// TwinCAT 3 PLC project UnitTest
// Title: UnitTest
// Company: Hoox.Software
// Author: Patrick Dressel
// ProjectVersion: 1.0.0
// ProgramVersion: 3.1.4022.6
// libraries:
//   Tc2_Standard, * (Beckhoff Automation GmbH)
//   Tc2_System, * (Beckhoff Automation GmbH)
//   Tc2_Utilities, * (Beckhoff Automation GmbH)
//   Tc3_Module, * (Beckhoff Automation GmbH)
//   Base Interfaces,newest,System
// project tree:
//   Datatypes/Coverage/ ALines_t.TcDUT, EReportType_t.TcDUT (not stored), SCodeCoverage_t.TcDUT (not stored)
//   Datatypes/ EResult_t.TcDUT (not stored), EState_t.TcDUT, IdHandle_t.TcDUT (not stored), ObjectId_t.TcDUT (not stored), SResult_t.TcDUT (not stored), SStatistic_t.TcDUT (not stored), StringHandle_t.TcDUT (not stored), StrMessage_t.TcDUT (not stored), TestCaseHandle_t.TcDUT (not stored), TestSuiteHandle_t.TcDUT
//   Datatypes/Report/ EExportState_t.TcDUT (not stored), ERetCode_t.TcDUT (not stored), NameHandle_t.TcDUT (not stored), PathHandle_t.TcDUT (not stored), StrFileName_t.TcDUT (not stored), StrPathName_t.TcDUT (not stored), TestReportHandle_t.TcDUT, UBaseTypes_t.TcDUT, UTime_t.TcDUT (not stored)
//   / PlcTask.TcTTO (not stored)
//   Source/ FB_Testsuite.TcPOU, FB_UnitTestBase.TcPOU, PRG_UnitTestLib.TcPOU
//   Source/Report/ FB_CoverageFile.TcPOU (not stored), FB_TestReportBase.TcPOU, FB_FileBase.TcPOU, FB_TextReport.TcPOU

// ---- Datatypes/Coverage/ALines_t.TcDUT
TYPE ALines_t : Array[1..1000] of BYTE; END_TYPE

// ---- Datatypes/EState_t.TcDUT
{attribute 'qualified_only'}
{attribute 'strict'}
TYPE EState_t :
(
	eStateInit,
	eStateIdle,
	eStatePrepare,
	eStateExecute,
	eStateCleanUp,
	eStateBuildCoverageFile,
	eStateBuildUnitTestFile,
	eStateReady,
	eStateExport,
	eStateError,
	eStateLicenseError
);
END_TYPE

// ---- Datatypes/Report/TestReportHandle_t.TcDUT
TYPE TestReportHandle_t : Pointer to FB_TestReportBase; END_TYPE

// ---- Datatypes/Report/UBaseTypes_t.TcDUT
TYPE UBaseTypes_t :
UNION
	u8Value 	: USINT;
	s8Value 	: SINT;
	u16Value 	: UINT;
	s16Value 	: INT;
	u32Value 	: UDINT;
	s32Value 	: DINT;
	w16Value    : WORD;
	w32Value    : DWORD;
END_UNION
END_TYPE

// ---- Datatypes/TestSuiteHandle_t.TcDUT
TYPE TestSuiteHandle_t : POINTER TO FB_TestSuite; END_TYPE

// ---- Source/FB_Testsuite.TcPOU
(******************************************************************************
Baustein: FB_Testsuite
Spezifikation: doc/Spezifikation.pdf, Kap. x.y.z
-------------------------------------------------------------------------------
erstellt:
von:
Geändert:
von:
-------------------------------------------------------------------------------
Beschreibung
Dieser Baustein enthält alle zugeordneten Testfälle. Ein Testfall
ist ein abgeleiteter Baustein (FB) von FB_UnitTestBase.

-------------------------------------------------------------------------------
Input
-

Output
-
******************************************************************************)
FUNCTION_BLOCK FB_Testsuite
VAR_INPUT
	i_bStart : BOOL;
END_VAR
VAR_OUTPUT
	o_eState  		: EState_t;
	o_eResult 		: EResult_t;
END_VAR
VAR
	strId			: ObjectId_t;
	strPath			: ObjectId_t;
	bRegistered     : BOOL;
	a_pTest  		: ARRAY [0..255] OF TestCaseHandle_t;
	pTest     		: TestCaseHandle_t;
	u16TestCases  	: UINT;
	u16Index 		: UINT;
	sStatistic 		: SStatistic_t;
END_VAR


	CASE o_eState OF
		
	EState_t.eStateInit:
	
		o_eState 	:= EState_t.eStateError;
		IF bRegistered = TRUE THEN
			o_eState 	:= EState_t.eStateIdle;
		END_IF;
		
	EState_t.eStateIdle:

		u16Index := 0;

		IF i_bStart = TRUE THEN
			logInfo(CONCAT('Run Testsuite ', strId));
			pTest 	 := getFirstTestCase();
			o_eState  := EState_t.eStatePrepare;
			o_eResult := EResult_t.eStatePassed;
		END_IF;

	EState_t.eStatePrepare:
	
		sStatistic.u32Executed  := 0;
		sStatistic.u32Passed 	:= 0;
		sStatistic.u32Failed 	:= 0;
		sStatistic.u32Asserts 	:= 0;

		IF pTest <> 0 THEN
			IF pTest^._prepare() = TRUE THEN
				pTest 	:= getNextTestCase();
			END_IF;
		ELSE
			o_eState := EState_t.eStateExecute;
			pTest 	:= getFirstTestCase();
		END_IF;

	EState_t.eStateExecute:

		IF pTest <> 0 THEN

			IF pTest^.isSkipped() = FALSE THEN

				pTest^.setStartTime();

				IF pTest^._execute() = TRUE THEN
					pTest^.setEndTime();
					sStatistic.u32Executed := sStatistic.u32Executed + 1;	
				
					sStatistic.u32Passed 	:= sStatistic.u32Passed + pTest^.getPassed();
					sStatistic.u32Failed 	:= sStatistic.u32Failed + pTest^.getFailed();
					sStatistic.u32Asserts   := sStatistic.u32Passed + sStatistic.u32Failed;
					
					CASE o_eResult OF 
	
					EResult_t.eStatePassed:
						// Status des letzen Tests übernehmen
						o_eResult := pTest^.o_eResult;
	
					EResult_t.eStateFailed:
						// Status nur übernehmen wenn ein Fatal-Status
						// ermittelt wird und der Test sofort abgebrochen
						// werden soll.
						IF pTest^.o_eResult = EResult_t.eStateFailedFatal THEN
							o_eResult := pTest^.o_eResult;
							o_eState  := EState_t.eStateCleanUp;
							pTest 	  := getFirstTestCase();	
						END_IF;
	
					EResult_t.eStateFailedFatal:
	
						o_eState := EState_t.eStateCleanUp;
						pTest 	:= getFirstTestCase();					
	
					END_CASE;
	
					IF o_eResult <> EResult_t.eStateFailedFatal THEN
						pTest 	 := getNextTestCase();
					END_IF;
	
				END_IF;
			ELSE
				pTest 	 := getNextTestCase();
			END_IF;
		ELSE
			o_eState := EState_t.eStateCleanUp;
			pTest 	:= getFirstTestCase();
		END_IF;

	ESTate_t.eStateCleanUp:

		IF pTest <> 0 THEN
			IF pTest^._cleanup() = TRUE THEN
				pTest 	:= getNextTestCase();
			END_IF;
		ELSE
			o_eState := EState_t.eStateReady;
		END_IF;
		
	ESTate_t.eStateReady:
	
		IF i_bStart = FALSE THEN
			o_eState := EState_t.eStateIdle;
		END_IF
		
	ESTate_t.eStateError:	
		
		// wenn wir hier rauskommen ist was dummes passiert
		
	ELSE
		
		o_eState := EState_t.eStateError;
		
	END_CASE;
	
	
	
	
	
	
//

(******************************************************************************
Baustein: FB_Testsuite.addTestcase
Spezifikation: doc/Spezifikation.pdf, Kap. x.y.z
-------------------------------------------------------------------------------
erstellt:
von:
Geändert:
von:
-------------------------------------------------------------------------------
Beschreibung
Diese Methode

-------------------------------------------------------------------------------
Input
i_pTestCase

Output
-
******************************************************************************)
{attribute 'hide'} 
METHOD PUBLIC addTestcase : BOOL
VAR_INPUT
	i_pTestCase : TestCaseHandle_t;
END_VAR

	addTestcase := FALSE;

	IF 	i_pTestCase  <> 0   AND 
		u16TestCases <  255 THEN
		
		a_pTest[u16TestCases] := i_pTestCase;
		
		u16TestCases := u16TestCases +1;
		
		sStatistic.u32TestCases := sStatistic.u32TestCases + 1;
		
		addTestcase := true;
	END_IF
END_METHOD

(******************************************************************************
Baustein: FB_Testsuite.FB_init
Spezifikation: doc/Spezifikation.pdf, Kap. x.y.z
-------------------------------------------------------------------------------
erstellt:
von:
Geändert:
von:
-------------------------------------------------------------------------------
Beschreibung
Diese Methode

-------------------------------------------------------------------------------
Input
i_pTestCase

Output
-
******************************************************************************)
{attribute 'hide'} 
METHOD FB_init : BOOL
VAR_INPUT
	bInitRetains 	: BOOL; // if TRUE, the retain variables are initialized (warm start / cold start)
	bInCopyCode 	: BOOL;  // if TRUE, the instance afterwards gets moved into the copy code (online change)
	i_strId	  		: ObjectId_t;
	i_strPath		: ObjectId_t;
END_VAR

	strId 	:= i_StrId;
	strPath := i_strPath;
	register();
END_METHOD

(******************************************************************************
Baustein: FB_Testsuite.getExecuted
Spezifikation: doc/Spezifikation.pdf, Kap. x.y.z
-------------------------------------------------------------------------------
erstellt:
von:
Geändert:
von:
-------------------------------------------------------------------------------
Beschreibung
Diese Methode

-------------------------------------------------------------------------------
Input
-

Output
-
******************************************************************************)
{attribute 'hide'} 
METHOD PUBLIC getExecuted : UDINT
VAR_INPUT
END_VAR

	getExecuted := sStatistic.u32Executed;
END_METHOD

(******************************************************************************
Baustein: FB_Testsuite.getFailed
Spezifikation: doc/Spezifikation.pdf, Kap. x.y.z
-------------------------------------------------------------------------------
erstellt:
von:
Geändert:
von:
-------------------------------------------------------------------------------
Beschreibung
Diese Methode

-------------------------------------------------------------------------------
Input
-

Output
-
******************************************************************************)
{attribute 'hide'} 
METHOD PUBLIC getFailed : UDINT
VAR_INPUT
END_VAR

	getFailed := sStatistic.u32Failed;
END_METHOD

(******************************************************************************
Baustein: FB_Testsuite.getFirstTestCase
Spezifikation: doc/Spezifikation.pdf, Kap. x.y.z
-------------------------------------------------------------------------------
erstellt:
von:
Geändert:
von:
-------------------------------------------------------------------------------
Beschreibung
Diese Methode

-------------------------------------------------------------------------------
Input
-

Output
-
******************************************************************************)
{attribute 'hide'} 
METHOD PUBLIC getFirstTestCase : TestCaseHandle_t
VAR_INPUT
END_VAR

	u16Index := 0;
	getFirstTestCase := a_pTest[0];
END_METHOD

(******************************************************************************
Baustein: FB_Testsuite.getId
Spezifikation: doc/Spezifikation.pdf, Kap. x.y.z
-------------------------------------------------------------------------------
erstellt:
von:
Geändert:
von:
-------------------------------------------------------------------------------
Beschreibung
Diese Methode

-------------------------------------------------------------------------------
Input
-

Output
-
******************************************************************************)
{attribute 'hide'} 
METHOD PUBLIC getId : STRING
VAR_INPUT
END_VAR

	getId := strId;
END_METHOD

(******************************************************************************
Baustein: FB_Testsuite.getNextTestCase
Spezifikation: doc/Spezifikation.pdf, Kap. x.y.z
-------------------------------------------------------------------------------
erstellt:
von:
Geändert:
von:
-------------------------------------------------------------------------------
Beschreibung
Diese Methode

-------------------------------------------------------------------------------
Input
-

Output
-
******************************************************************************)
{attribute 'hide'} 
METHOD PUBLIC getNextTestCase : TestCaseHandle_t
VAR_INPUT
END_VAR

	getNextTestCase := 0;
	u16Index 		 := u16Index + 1;

	IF u16Index < u16TestCases THEN
		getNextTestCase := a_pTest[u16Index];
	END_IF;
END_METHOD

(******************************************************************************
Baustein: FB_Testsuite.getNoOfAsserts
Spezifikation: doc/Spezifikation.pdf, Kap. x.y.z
-------------------------------------------------------------------------------
erstellt:
von:
Geändert:
von:
-------------------------------------------------------------------------------
Beschreibung
Diese Methode

-------------------------------------------------------------------------------
Input
-

Output
-
******************************************************************************)
{attribute 'hide'} 
METHOD PUBLIC getNoOfAsserts : UDINT
VAR_INPUT
END_VAR

	getNoOfAsserts := sStatistic.u32Asserts;
END_METHOD

(******************************************************************************
Baustein: FB_Testsuite.getNoOfTests
Spezifikation: doc/Spezifikation.pdf, Kap. x.y.z
-------------------------------------------------------------------------------
erstellt:
von:
Geändert:
von:
-------------------------------------------------------------------------------
Beschreibung
Diese Methode

-------------------------------------------------------------------------------
Input
-

Output
-
******************************************************************************)
{attribute 'hide'} 
METHOD PUBLIC getNoOfTests : UDINT
VAR_INPUT
END_VAR

	getNoOfTests := sStatistic.u32TestCases;
END_METHOD

(******************************************************************************
Baustein: FB_Testsuite.getPassed
Spezifikation: doc/Spezifikation.pdf, Kap. x.y.z
-------------------------------------------------------------------------------
erstellt:
von:
Geändert:
von:
-------------------------------------------------------------------------------
Beschreibung
Diese Methode

-------------------------------------------------------------------------------
Input
-

Output
-
******************************************************************************)
{attribute 'hide'} 
METHOD PUBLIC getPassed : UDINT
VAR_INPUT
END_VAR

	getPassed := sStatistic.u32Passed;
END_METHOD

{attribute 'hide'} 
METHOD PUBLIC getPath : ObjectId_t
VAR_INPUT
END_VAR

	getPath := strPath;
END_METHOD

(******************************************************************************
Baustein: FB_Testsuite.logInfo
Spezifikation: doc/Spezifikation.pdf, Kap. x.y.z
-------------------------------------------------------------------------------
erstellt:
von:
Geändert:
von:
-------------------------------------------------------------------------------
Beschreibung
Diese Methode

-------------------------------------------------------------------------------
Input
i_strMessage

Output
-
******************************************************************************)
{attribute 'hide'} 
METHOD PROTECTED logInfo : BOOL
VAR_INPUT
	i_strMessage : StrMessage_t;
END_VAR

	ADSLOGSTR(msgCtrlMask 	:= ADSLOG_MSGTYPE_HINT , 
			  msgFmtStr 	:= i_strMessage, 
			  strArg 		:= '');
END_METHOD

(******************************************************************************
Baustein: FB_Testsuite.register
Spezifikation: doc/Spezifikation.pdf, Kap. x.y.z
-------------------------------------------------------------------------------
erstellt:
von:
Geändert:
von:
-------------------------------------------------------------------------------
Beschreibung
Diese Methode

-------------------------------------------------------------------------------
Input
-

Output
-
******************************************************************************)
{attribute 'hide'} 
METHOD PROTECTED register : BOOL
VAR_INPUT
END_VAR

	bRegistered := PRG_UnitTestLib.addTestSuite(this);
END_METHOD

END_FUNCTION_BLOCK

// ---- Source/PRG_UnitTestLib.TcPOU
(******************************************************************************
Baustein: PRG_TestLibrary
Spezifikation: doc/Spezifikation.pdf, Kap. x.y.z
-------------------------------------------------------------------------------
erstellt:
von:
Geändert:
von:
-------------------------------------------------------------------------------
Beschreibung
Dieser Baustein etnhält alle Testsuites und führt diese aus.

-------------------------------------------------------------------------------
Input
	i_bStart : mit positiver Flanke werden die registrierten Testsuites ausgeführt

Output
	o_eState  		: EState_t;
	o_eResult 		: EResult_t;
	o_sStatistic	: SStatistic_t;
******************************************************************************)
{attribute 'global_init_slot' := '41000'}
PROGRAM PRG_UnitTestLib
VAR_INPUT
	i_bStart : BOOL;
END_VAR
VAR_OUTPUT
	o_eState  		: EState_t;
	o_eResult 		: EResult_t;
	o_sStatistic	: SStatistic_t;
END_VAR
VAR
	a_pTestSuite 	: ARRAY [0..255] OF TestSuiteHandle_t;
	u16TestSuites 	: UINT;
	u16Index	  	: UINT;
	pActTestSuite 	: TestSuiteHandle_t;
	pTestReport		: POINTER TO FB_TestReportBase;
	eRetCode 		: ERetCode_t;

	fbSystemTime 	: FB_LocalSystemTime;
	
	fbLicense 		: FB_CheckLicense;
	
	
	fbCoverage 		: FB_CoverageFile;
	fbUnittest 		: FB_CoverageFile;
	u16PouIdx  		: UINT;
	u16LineIdx 		: UINT;
	u16ReportState  : UINT;
	u16TestSuitIdx	: UINT;
	sCodeCoverage	: SCodeCoverage_t;
	pTestCase  		: TestCaseHandle_t;
END_VAR


	fbSystemTime(bEnable := TRUE, dwCycle := 5);

	fbCoverage();

	fbUnittest();

	CASE o_eState OF 
	
	EState_t.eStateInit:	

		//IF checkLicense() = ERetCode_t.eRetDone THEN
			
			IF i_bStart = FALSE THEN 
				o_eState := EState_t.eStateIdle; 
			END_IF
			
		//END_IF;
	
	EState_t.eStateIdle:
	
		IF i_bStart = TRUE THEN
			logInfo('+++++++++++++ Testbeginn ++++++++++++++');
			o_eState := EState_t.eStatePrepare;
		END_IF
	
	EState_t.eStatePrepare:
		
		o_eResult 	  				:= EResult_t.eStatePassed;
		o_sStatistic.u32Executed 	:= 0;
		o_sStatistic.u32TestCases	:= 0;
		o_sStatistic.u32Asserts  	:= 0;
		o_sStatistic.u32Passed   	:= 0;
		o_sStatistic.u32Failed	 	:= 0;	

		pActTestSuite := getFirstTestSuite();
		
		IF pActTestSuite      <> 0   THEN
			o_eState := EState_t.eStateExecute;
		ELSE
			o_eState := EState_t.eStateError;	
		END_IF
	
	EState_t.eStateExecute:
	
		pActTestSuite^(i_bStart := TRUE);
	
		IF pActTestSuite^.o_eState = EState_t.eStateReady THEN
			
			IF pActTestSuite^.o_eResult = EResult_t.eStateFailed THEN
				o_eResult := EResult_t.eStateFailed;
			END_IF
			
			pActTestSuite^(i_bStart := FALSE);
			
			o_eState := EState_t.eStateCleanUp;
			
			o_sStatistic.u32Executed 	:= o_sStatistic.u32Executed  + pActTestSuite^.getExecuted();
			o_sStatistic.u32TestCases	:= o_sStatistic.u32TestCases + pActTestSuite^.getNoOfTests(); 
			o_sStatistic.u32Asserts  	:= o_sStatistic.u32Asserts   + pActTestSuite^.getNoOfAsserts();
			o_sStatistic.u32Passed   	:= o_sStatistic.u32Passed    + pActTestSuite^.getPassed();
			o_sStatistic.u32Failed	 	:= o_sStatistic.u32Failed    + pActTestSuite^.getFailed();
		END_IF
	
	EState_t.eStateCleanUp:
	
		IF pActTestSuite^.o_eResult = EResult_t.eStateFailedFatal THEN
			o_eResult := EResult_t.eStateFailedFatal;
			o_eState  := EState_t.eStateBuildCoverageFile;
		ELSE
			
			pActTestSuite := getNextTestSuite();
						
			IF pActTestSuite <> 0 THEN
				o_eState := EState_t.eStateExecute;
			ELSE
				o_eState := EState_t.eStateBuildCoverageFile;
				logInfo('+++++++++++++ Test Ende ++++++++++++++');
			END_IF		
			
		END_IF

	EState_t.eStateBuildCoverageFile:

		IF createReport(EReporttype_t.eCoverageReport) = ERetCode_t.eRetDone THEN
			o_eState := EState_t.eStateBuildUnitTestFile;
		END_IF;

	EState_t.eStateBuildUnitTestFile:

		IF createReport(EReporttype_t.eUnitTestReport) = ERetCode_t.eRetDone THEN
			o_eState := EState_t.eStateReady;
		END_IF;

	EState_t.eStateReady:

		IF i_bStart = FALSE THEN
			o_eState := EState_t.eStateExport;
		END_IF

	EState_t.eStateExport:

		IF createReport(EReporttype_t.eExternalReport) = ERetCode_t.eRetDone THEN
			o_eState := EState_t.eStateIdle;
		END_IF;

	EState_t.eStateError,
	EState_t.eStateLicenseError:
	
		o_eState := EState_t.eStateError;

	END_CASE

(******************************************************************************
Baustein: PRG_UnitTestLib.addTestReport
Spezifikation: doc/Spezifikation.pdf, Kap. x.y.z
-------------------------------------------------------------------------------
erstellt:
von:
Geändert:
von:
-------------------------------------------------------------------------------
Beschreibung
Diese Methode

-------------------------------------------------------------------------------
Input
i_pTestReport

Output
-
******************************************************************************)
{attribute 'hide'} 
METHOD PUBLIC addTestReport : BOOL
VAR_INPUT
	i_pTestReport : TestReportHandle_t;
END_VAR

	pTestReport := i_pTestReport;
END_METHOD

(******************************************************************************
Baustein: PRG_UnitTestLib.addTestSuite
Spezifikation: doc/Spezifikation.pdf, Kap. x.y.z
-------------------------------------------------------------------------------
erstellt:
von:
Geändert:
von:
-------------------------------------------------------------------------------
Beschreibung
Diese Methode

-------------------------------------------------------------------------------
Input
i_pTestSuite

Output
-
******************************************************************************)
{attribute 'hide'} 
METHOD PUBLIC addTestSuite : BOOL
VAR_INPUT
	i_pTestSuite : TestSuiteHandle_t;
END_VAR

	addTestSuite := FALSE;

	IF 	i_pTestSuite  <> 0   AND 
		u16TestSuites <  255 THEN
		
		a_pTestSuite[u16TestSuites] := i_pTestSuite;
		
		u16TestSuites := u16TestSuites +1;
	
		o_sStatistic.u32TestSuites := o_sStatistic.u32TestSuites + 1;
		o_sStatistic.u32TestCases  := o_sStatistic.u32TestCases + i_pTestSuite^.sStatistic.u32TestCases;
		
		addTestSuite := TRUE;
	END_IF
END_METHOD

(******************************************************************************
Baustein: PRG_UnitTestLib.checkLicense
Spezifikation: doc/Spezifikation.pdf, Kap. x.y.z
-------------------------------------------------------------------------------
erstellt:
von:
Geändert:
von:
-------------------------------------------------------------------------------
Beschreibung
Diese Methode

-------------------------------------------------------------------------------
Input
-

Output
-
******************************************************************************)
{attribute 'hide'} 
METHOD checkLicense : ERetCode_t
VAR_INPUT
END_VAR

	checkLicense := ERetCode_t.eRetBusy;
	
	fbLicense(bExecute    := TRUE, 
		  stLicenseId := STRING_TO_GUID('994D9F0C-F802-4000-8582-229354A3CA39'));
			  
	IF fbLicense.bBusy =  FALSE THEN
		IF fbLicense.stCheckLicense.eResult = E_LHR_LicenseOK THEN
			checkLicense := ERetCode_t.eRetDone;
		ELSE
			checkLicense := ERetCode_t.eRetFailed;	
		END_IF
	END_IF;
END_METHOD

{attribute 'hide'} 
METHOD PRIVATE createReport : ERetCode_t
VAR_INPUT
	i_eReporttype : EReportType_t;
END_VAR
VAR
	eRetcode : ERetCode_t;
	u32Temp : UDINT;
END_VAR

	createReport := ERetCode_t.eRetBusy;

	CASE u16ReportState OF

	0: 
		IF i_eReporttype = EReportType_t.eCoverageReport THEN
			u16ReportState := 10;
		END_IF;

		IF i_eReporttype = EReportType_t.eUnitTestReport THEN
			u16ReportState := 20;
		END_IF;

		IF i_eReporttype = EReportType_t.eExternalReport THEN
			u16ReportState := 100;
		END_IF;

// +++++++++++++++++++++++++++++++++++++++++++++++++++++++++++
//
// Export Codeabdeckung
// 
// +++++++++++++++++++++++++++++++++++++++++++++++++++++++++++
	10:
		eRetcode := fbCoverage.open('C:\Users\Administrator\Desktop\TestResult\', 'Coverage.xml');

		IF eRetcode = ERetCode_t.eRetDone THEN

			u16ReportState := 11;

		ELSIF eRetcode = ERetCode_t.eRetFailed THEN

			logError('createReport Coverage.xml : Datei nicht geöffnet');
			u16ReportState := 12;

		END_IF;		

	11:

		fbCoverage.addString('<?xml version="1.0" ?>');
		fbCoverage.addCrlf();

		fbCoverage.addString('<Result>');
		fbCoverage.addCrlf();

		FOR u16PouIdx := 1 TO sCodeCoverage.u16MaxIndex DO

			fbCoverage.addString('<POU Id="');
			fbCoverage.addValue(u16PouIdx);
			fbCoverage.addString('">');
			fbCoverage.addCrlf();

			FOR u16LineIdx := 1 TO 1000 DO

				IF sCodeCoverage.aPou[u16PouIdx][u16LineIdx] > 0 THEN

					fbCoverage.addString('<Line Nb="');
					fbCoverage.addValue(u16LineIdx);

					fbCoverage.addString('" Count="');
					fbCoverage.addValue(sCodeCoverage.aPou[u16PouIdx][u16LineIdx]);
					
					fbCoverage.addString('"/>');
					fbCoverage.addCrlf();

				END_IF;

			END_FOR;

			fbCoverage.addString('</POU>');
			fbCoverage.addCrlf();

		END_FOR;

		fbCoverage.addString('</Result>');
		fbCoverage.addCrlf();
		u16ReportState := 12;


	12:

		IF fbCoverage.o_bOpen  = TRUE AND 
		   fbCoverage.o_bEmpty = TRUE THEN
			fbCoverage.close();
		END_IF;

		IF fbCoverage.o_bOpen  = FALSE THEN
			createReport 	:= ERetCode_t.eRetDone;
		END_IF;

// +++++++++++++++++++++++++++++++++++++++++++++++++++++++++++
//
// Export Unittest Ergebnisse
// 
// +++++++++++++++++++++++++++++++++++++++++++++++++++++++++++
	20:		

		eRetcode := fbUnitTest.open('C:\Users\Administrator\Desktop\TestResult\', 'Unittest.xml');

		IF eRetcode = ERetCode_t.eRetDone THEN

			u16ReportState := 21;

		ELSIF eRetcode = ERetCode_t.eRetFailed THEN

			logError('createReport Unittest.xml : Datei nicht geöffnet');
			u16ReportState := 22;

		END_IF;	

	21:

		u16TestSuitIdx := 0;

		fbUnitTest.addString('<?xml version="1.0" ?>');
		fbUnitTest.addCrlf();

		fbUnitTest.addString('<testsuites>');
		fbUnitTest.addCrlf();

		pActTestSuite := getFirstTestSuite();

		WHILE (pActTestSuite <> 0) DO

			u16TestSuitIdx := u16TestSuitIdx+1;

			fbUnitTest.addString('<testsuite');
			fbUnitTest.addString(' name="');
			fbUnitTest.addString(pActTestSuite^.getId());
			fbUnitTest.addString('" tests="');
			u32Temp := pActTestSuite^.getNoOfTests();
			fbUnitTest.addValue(u32Temp);
			fbUnitTest.addString('" disabled="');
			u32Temp := 0;
			fbUnitTest.addValue(u32Temp);
			fbUnitTest.addString('" errors="');
			fbUnitTest.addValue(u32Temp);
			fbUnitTest.addString('" failures="');
			u32Temp := pActTestSuite^.getFailed();
			fbUnitTest.addValue(u32Temp);
			fbUnitTest.addString('" hostname="');
			fbUnitTest.addString('" id="');
			fbUnitTest.addvalue(u16TestSuitIdx);
			fbUnitTest.addString('" package="');
			fbUnitTest.addString(pActTestSuite^.getPath());
			fbUnitTest.addString('">');
			fbUnitTest.addCrlf();

			pTestCase := pActTestSuite^.getFirstTestCase();

			WHILE (pTestCase <> 0) DO

				fbUnitTest.addString('<testcase');
				fbUnitTest.addString(' name="');
				fbUnitTest.addString(pTestCase^.getId());
				fbUnitTest.addString('" assertions="');
				u32Temp := pTestCase^.getFailed() + pTestCase^.getPassed();
				fbUnitTest.addValue(u32Temp);
				fbUnitTest.addString('" classname="');
				fbUnitTest.addString(pTestCase^.getPath());
				fbUnitTest.addString(pTestCase^.getClassName());
				fbUnitTest.addString('" time="');
				u32Temp := pTestCase^.getTime();
				fbUnitTest.addTimeMs(u32Temp);
				fbUnitTest.addString('">');
				fbUnitTest.addCrlf();

				CASE pTestCase^.o_eResult OF

				EResult_t.eStatePassed :

					fbUnitTest.addString('<passed/>');

				EResult_t.eStateFailed, 
				EResult_t.eStateFailedFatal :
			
					fbUnitTest.addString('<failure/>');

				EResult_t.eStateSkipped:

					fbUnitTest.addString('<skipped/>');

				END_CASE;
				
				fbUnitTest.addCrlf();	

				fbUnitTest.addString('</testcase>');
				fbUnitTest.addCrlf();		

				pTestCase := pActTestSuite^.getNextTestCase();
		
			END_WHILE

			fbUnitTest.addString('</testsuite>');
			fbUnitTest.addCrlf();	

			pActTestSuite := getNextTestSuite();

		END_WHILE

		fbUnitTest.addString('</testsuites>');
		fbUnitTest.addCrlf();

		u16ReportState := 22;

	22:
		IF fbUnitTest.o_bOpen  = TRUE AND 
		   fbUnitTest.o_bEmpty = TRUE THEN
			fbUnitTest.close();
		END_IF;

		IF fbUnitTest.o_bOpen  = FALSE THEN
			createReport 	:= ERetCode_t.eRetDone;
		END_IF;

// +++++++++++++++++++++++++++++++++++++++++++++++++++++++++++
//
//
// 
// +++++++++++++++++++++++++++++++++++++++++++++++++++++++++++
	100:

		IF pTestReport <> 0 THEN
			
			createReport := pTestReport^.create();		
			
		ELSE

			createReport := ERetCode_t.eRetDone;

		END_IF;

	ELSE
		createReport := ERetCode_t.eRetFailed;
	END_CASE;

	IF createReport = ERetCode_t.eRetDone THEN
		u16ReportState := 0;
	END_IF;
















(**)
END_METHOD

(******************************************************************************
Baustein: PRG_UnitTestLib.getFirstTestSuite
Spezifikation: doc/Spezifikation.pdf, Kap. x.y.z
-------------------------------------------------------------------------------
erstellt:
von:
Geändert:
von:
-------------------------------------------------------------------------------
Beschreibung
Diese Methode

-------------------------------------------------------------------------------
Input
-

Output
-
******************************************************************************)
{attribute 'hide'} 
METHOD PRIVATE getFirstTestSuite : TestSuiteHandle_t
VAR_INPUT
END_VAR

	u16Index := 0;
	getFirstTestSuite := a_pTestSuite[0];
END_METHOD

(******************************************************************************
Baustein: PRG_UnitTestLib.getNextTestSuite
Spezifikation: doc/Spezifikation.pdf, Kap. x.y.z
-------------------------------------------------------------------------------
erstellt:
von:
Geändert:
von:
-------------------------------------------------------------------------------
Beschreibung
Diese Methode

-------------------------------------------------------------------------------
Input
-

Output
-
******************************************************************************)
{attribute 'hide'} 
METHOD PRIVATE getNextTestSuite : TestSuiteHandle_t
VAR_INPUT
END_VAR

	getNextTestSuite := 0;
	u16Index 		 := u16Index + 1;

	IF u16Index < u16TestSuites THEN
		getNextTestSuite := a_pTestSuite[u16Index];
	END_IF;
END_METHOD

(******************************************************************************
Baustein: PRG_UnitTestLib.getTime
Spezifikation: doc/Spezifikation.pdf, Kap. x.y.z
-------------------------------------------------------------------------------
erstellt:
von:
Geändert:
von:
-------------------------------------------------------------------------------
Beschreibung
Diese Methode

-------------------------------------------------------------------------------
Input
-

Output
-
******************************************************************************)
{attribute 'hide'} 
METHOD getTime : TimeStruct
VAR_INPUT
END_VAR
VAR
END_VAR

	getTime := fbSystemTime.systemTime;
END_METHOD

{attribute 'hide'} 
METHOD PUBLIC LineCovered : BOOL
VAR_INPUT
	u16Pou  : UINT;
	u16Line : UINT;
END_VAR

	LineCovered := TRUE;
	
	IF o_eState = EState_t.eStateExecute THEN

		IF (u16Pou  > 0 AND u16Pou  <= 2000) AND
           (u16Line > 0 AND u16Line <= 1000) THEN

			IF u16Pou > sCodeCoverage.u16MaxIndex THEN
				sCodeCoverage.u16MaxIndex := u16Pou;
			END_IF;

			IF sCodeCoverage.aPou[u16Pou][u16Line] < 255 THEN
				sCodeCoverage.aPou[u16Pou][u16Line] := sCodeCoverage.aPou[u16Pou][u16Line]+1;
			END_IF;
		END_IF;

	END_IF;
END_METHOD

(******************************************************************************
Baustein: PRG_UnitTestLib.logError
Spezifikation: doc/Spezifikation.pdf, Kap. x.y.z
-------------------------------------------------------------------------------
erstellt:
von:
Geändert:
von:
-------------------------------------------------------------------------------
Beschreibung
Diese Methode

-------------------------------------------------------------------------------
Input
i_strMessage

Output
-
******************************************************************************)
{attribute 'hide'} 
METHOD PROTECTED logError : BOOL
VAR_INPUT
	i_strMessage : StrMessage_t;
END_VAR

	ADSLOGSTR(msgCtrlMask 	:= ADSLOG_MSGTYPE_ERROR , 
			  msgFmtStr 	:= i_strMessage, 
			  strArg 		:= '');
END_METHOD

(******************************************************************************
Baustein: PRG_UnitTestLib.logInfo
Spezifikation: doc/Spezifikation.pdf, Kap. x.y.z
-------------------------------------------------------------------------------
erstellt:
von:
Geändert:
von:
-------------------------------------------------------------------------------
Beschreibung
Diese Methode

-------------------------------------------------------------------------------
Input
i_strMessage

Output
-
******************************************************************************)
{attribute 'hide'} 
METHOD PUBLIC logInfo : BOOL
VAR_INPUT
	i_strMessage : StrMessage_t;
END_VAR

	ADSLOGSTR(msgCtrlMask 	:= ADSLOG_MSGTYPE_HINT , 
			  msgFmtStr 	:= i_strMessage, 
			  strArg 		:= '');
END_METHOD

END_PROGRAM

// ---- Source/Report/FB_TestReportBase.TcPOU
(******************************************************************************
Baustein: FB_TestReportBase
Spezifikation: doc/Spezifikation.pdf, Kap. x.y.z
-------------------------------------------------------------------------------
erstellt:
von:
Geändert:
von:
-------------------------------------------------------------------------------
Beschreibung
Dieser Baustein enthält alle zugeordneten Testfälle. Ein Testfall
ist ein abgeleiteter Baustein (FB) von FB_UnitTestBase.

-------------------------------------------------------------------------------
Input
-

Output
-
******************************************************************************)
FUNCTION_BLOCK FB_TestReportBase
VAR_INPUT
END_VAR
VAR_OUTPUT
END_VAR
VAR
	strBuffer   : STRING(255);
	fbOpen      : FB_FileOpen;
	fbClose     : FB_FileClose;
	fbWrite	    : FB_FileWrite;
	strFileName : StrFileName_t;
	strFilePath : StrPathName_t;
	
	eState 		: EExportState_t;
	u32Line     : UDINT;
	
	sStatistic  : SStatistic_t;

	trgOpen 	: F_TRIG;
	trgWrite 	: F_TRIG;
	trgClose 	: F_TRIG;
END_VAR

METHOD PROTECTED addCrlf : BOOL
VAR_INPUT
END_VAR
VAR
END_VAR
   
	strBuffer := CONCAT(strBuffer, '$R$N');
END_METHOD

METHOD PROTECTED addDate : ERetCode_t
VAR_INPUT
	i_sDate : TIMESTRUCT;
END_VAR

   	addDate := ERetcode_t.eRetDone;

   	addValue(i_sDate.wDay);
   	addString('.');
   	addValue(i_sDate.wMonth);
   	addString('.');
    addValue(i_sDate.wYear);
    addString(' ');
END_METHOD

METHOD PROTECTED addString : ERetCode_t
VAR_INPUT
	i_strData : STRING(255);
END_VAR

	strBuffer :=  concat(strBuffer, i_strData);

	addString := ERetcode_t.eRetDone;
END_METHOD

METHOD PROTECTED addTime : ERetCode_t
VAR_INPUT
	i_sTime : TIMESTRUCT;
END_VAR

	addTime := ERetcode_t.eRetDone;
	
   	addValue(i_sTime.wHour);
   	addString('.');
   	addValue(i_sTime.wMinute);
  	addString('.');
   	addValue(i_sTime.wSecond);
   	addString(' ');
END_METHOD

METHOD PROTECTED addValue : ERetCode_t
VAR_INPUT
	i_anyValue : ANY;
END_VAR
VAR
	uValue : UBaseTypes_t;
END_VAR

	addValue  := ERetcode_t.eRetDone;
	
	IF i_anyValue.pValue = 0 THEN
		addValue  := ERetcode_t.eRetFailed;
		RETURN;
	END_IF

	MEMCPY(ADR(uValue),i_anyValue.pValue, TO_UDINT(i_anyValue.diSize)); 

	CASE i_anyValue.TypeClass OF

	IBaseLibrary.TYPE_SINT:

		addString(SINT_TO_STRING(uValue.s8Value));

	//IBaseLibrary.TYPE_BYTE:
	IBaseLibrary.TYPE_USINT:

		addString(USINT_TO_STRING(uValue.u8Value));

	IBaseLibrary.TYPE_INT:

		addString(INT_TO_STRING(uValue.s16Value));

	IBaseLibrary.TYPE_DINT:

		addString(DINT_TO_STRING(uValue.s32Value));

	IBaseLibrary.TYPE_UINT:

		addString(UINT_TO_STRING(uValue.u16Value));

	IBaseLibrary.TYPE_UDINT:

		addString(UDINT_TO_STRING(uValue.u32Value));

	IBaseLibrary.TYPE_WORD:

		addString(WORD_TO_STRING(uValue.w16Value));

	IBaseLibrary.TYPE_DWORD:

		addString(DWORD_TO_STRING(uValue.w32Value));

	ELSE
		ADSLOGSTR(msgCtrlMask 	:= ADSLOG_MSGTYPE_ERROR , 
				  msgFmtStr 	:= 'TestReportBase.AddValue: Unbekannter Datentyp!', 
				  strArg 		:= '');
	END_CASE;
END_METHOD

(******************************************************************************
Baustein: FB_TestReportBase.BuildFile
Spezifikation: doc/Spezifikation.pdf, Kap. x.y.z
-------------------------------------------------------------------------------
erstellt:
von:
Geändert:
von:
-------------------------------------------------------------------------------
Beschreibung
Diese Methode muss vom ableitenden Baustein überschrieben werden und
wird von der Basisklasse aus aufgerufen wenn der Report erstellt werden
soll.

-------------------------------------------------------------------------------
Input
-

Output
-
******************************************************************************)
METHOD PROTECTED BuildFile : ERetCode_t
VAR_INPUT
	i_u32Line : UDINT;
END_VAR
END_METHOD

METHOD PROTECTED clearBuffer : ERetCode_t
VAR_INPUT
END_VAR

	clearBuffer := ERetCode_t.eRetDone;
	
	strBuffer := '';
END_METHOD

METHOD PROTECTED Close : ERetCode_t
VAR_INPUT
END_VAR

	Close := ERetCode_t.eRetFailed;
	
	fbClose.hFile 		:= fbOpen.hFile;
	fbClose.bExecute 	:= TRUE; 

	IF trgClose.Q = TRUE THEN
		Close := ERetCode_t.eRetDone;
		fbClose.bExecute  := FALSE;		
	ELSE	
		Close := ERetCode_t.eRetBusy;
	END_IF;	
	
	IF fbClose.bError = TRUE THEN
		Close := eRetCode_t.eRetFailed;
	END_IF;
END_METHOD

METHOD PUBLIC create : ERetCode_t;
VAR_INPUT
END_VAR
VAR
	eRetCode : ERetCode_t;
END_VAR

	create := ERetCode_t.eRetBusy;

	fbOpen();
	fbWrite();
	fbClose();

	trgOpen(CLK := fbOpen.bBusy);
	trgWrite(CLK := fbWrite.bBusy);
	trgClose(CLK := fbClose.bBusy);
	
	CASE eState OF
	
	EExportState_t.eExportIdle:
	
		eState := EExportState_t.eExportOpen;
	
	EExportState_t.eExportOpen:
	
		eRetCode 	:= Open();
		u32Line  	:= 0;
		sStatistic 	:= PRG_UnitTestLib.o_sStatistic;

		IF eRetCode = ERetCode_t.eRetDone THEN
			eState := EExportState_t.eExportGetLine;
		ELSIF eRetCode = ERetCode_t.eRetFailed THEN
			eState := EExportState_t.eExportError;
		END_IF;

	EExportState_t.eExportGetLine:

		eRetCode := BuildFile(u32Line);

		IF eRetCode = ERetCode_t.eRetDone THEN
			eState := EExportState_t.eExportClose;
		ELSIF eRetCode = ERetCode_t.eRetFailed THEN
			eState := EExportState_t.eExportError;
		ELSE
			addCrlf();
			eState := EExportState_t.eExportWrite;
		END_IF;

	EExportState_t.eExportWrite:
	
		IF writeBuffer() =  ERetCode_t.eRetDone THEN
			clearBuffer();	
			u32Line := u32Line + 1;
			eState  := EExportState_t.eExportGetLine;
		END_IF;		
	
	EExportState_t.eExportClose:
	
		eRetCode := Close();
		
		IF eRetCode = ERetCode_t.eRetDone THEN
			eState     := EExportState_t.eExportIdle;
			create	   := ERetCode_t.eRetDone;
			reset();
		ELSIF eRetCode = ERetCode_t.eRetFailed THEN
			eState := EExportState_t.eExportError;
		end_if;
	
	EExportState_t.eExportError:
	
		create := ERetCode_t.eRetFailed;
	
	end_case;
END_METHOD

METHOD FB_init : BOOL
VAR_INPUT
	bInitRetains : BOOL; // if TRUE, the retain variables are initialized (warm start / cold start)
	bInCopyCode : BOOL;  // if TRUE, the instance afterwards gets moved into the copy code (online change)
END_VAR

	PRG_UnitTestLib.addTestReport(this);
END_METHOD

(******************************************************************************
Baustein: FB_TestReportBase.getFileName
Spezifikation: doc/Spezifikation.pdf, Kap. x.y.z
-------------------------------------------------------------------------------
erstellt:
von:
Geändert:
von:
-------------------------------------------------------------------------------
Beschreibung
Diese Methode muss vom ableitenden Baustein überschrieben werden und
wird von der Basisklasse aus aufgerufen wenn der Report erstellt werden
soll.

-------------------------------------------------------------------------------
Input
-

Output
-
******************************************************************************)
METHOD PROTECTED getFileName : ERetCode_t
VAR_INPUT
	i_pFileName : NameHandle_t;
	i_pPath		: PathHandle_t;
END_VAR
END_METHOD

METHOD PROTECTED getTime : TimeStruct
VAR_INPUT
END_VAR
VAR
END_VAR

	getTime := PRG_UnitTestLib.getTime();
END_METHOD

METHOD PROTECTED open : ERetCode_t
VAR_INPUT
END_VAR

	open := ERetCode_t.eRetFailed;

	getFileName(ADR(strFileName), ADR(strFilePath));
	
	fbOpen.sPathName := CONCAT(strFilePath, strFileName);
	fbOpen.nMode 	 := FOPEN_MODEWRITE OR FOPEN_MODEBINARY;	
	fbOpen.bExecute  := TRUE;
			
	IF trgOpen.Q = TRUE THEN
		open := ERetCode_t.eRetDone;
		fbOpen.bExecute  := FALSE;		
	ELSE	
		open := ERetCode_t.eRetBusy;
	END_IF;	
	
	IF fbOpen.bError = TRUE THEN
		open := eRetCode_t.eRetFailed;
	END_IF;
END_METHOD

METHOD PUBLIC reset : BOOL
VAR_INPUT
END_VAR

	IF fbOpen.hFile <> 0 THEN
		close();
	END_IF
	
	clearBuffer();

	fbOpen(sPathName := '', bExecute := FALSE);
	
	fbWrite(bExecute := FALSE);
	
	fbClose(bExecute := FALSE);
	
	eState := EExportState_t.eExportIdle;
END_METHOD

METHOD PROTECTED writeBuffer : ERetCode_t
VAR_INPUT
END_VAR
VAR
	u32Len : UDINT;
END_VAR

	writeBuffer := eRetCode_t.eRetBusy;
	
	IF LEN(strBuffer) <= 0 THEN
		RETURN;
	END_IF
	
	u32Len := TO_UDINT(LEN(strBuffer)); 
	
	writeBuffer := writeData(i_pData := ADR(strBuffer), u32Size := u32Len);
END_METHOD

METHOD PROTECTED writeData : ERetCode_t
VAR_INPUT
	i_pData : POINTER TO BYTE;
	u32Size : UDINT;
END_VAR

	writeData := ERetCode_t.eRetFailed;
	
	IF u32Size = 0 OR i_pData = 0 THEN
		RETURN;
	END_IF
	
	fbWrite.pWriteBuff 	:= i_pData; 
	fbWrite.cbWriteLen 	:= u32Size; 
	fbWrite.hFile 		:= fbOpen.hFile; 
	fbWrite.bExecute 	:= TRUE;
			
	IF trgWrite.Q = TRUE THEN
		writeData := ERetCode_t.eRetDone;
		fbWrite.bExecute 	:= FALSE;			
	ELSE	
		writeData := ERetCode_t.eRetBusy;
	END_IF;	

	IF fbWrite.bError = TRUE THEN
		writeData := eRetCode_t.eRetFailed;
	END_IF;
END_METHOD

END_FUNCTION_BLOCK

// ---- Source/FB_UnitTestBase.TcPOU
(******************************************************************************
Baustein: FB_UnitTestBase
Spezifikation: doc/Spezifikation.pdf, Kap. x.y.z
-------------------------------------------------------------------------------
erstellt:
von:
Geändert:
von:
-------------------------------------------------------------------------------
Beschreibung
Dieser Baustein stellt die Basis für einen Unittest dar und enthält
alle notwendigen Variablen und Methoden zur Testauswertung.

-------------------------------------------------------------------------------
Input
-

Output
	o_eState : EState_t;
	o_eResult: EResult_t;
******************************************************************************)
FUNCTION_BLOCK FB_UnitTestBase
VAR_INPUT
END_VAR
VAR_OUTPUT
	o_eState : EState_t;
	o_eResult: EResult_t;
END_VAR
VAR
	strId	  		: ObjectId_t;
	pTestSuite      : TestSuiteHandle_t;
	bRegistered 	: BOOL;
	u32Passed 		: UDINT;
	u32Failed 		: UDINT;
END_VAR

(******************************************************************************
Baustein: FB_UnitTestBase.addFailed
Spezifikation: doc/Spezifikation.pdf, Kap. x.y.z
-------------------------------------------------------------------------------
erstellt:
von:
Geändert:
von:
-------------------------------------------------------------------------------
Beschreibung
Diese Methode

-------------------------------------------------------------------------------
Input
-

Output
-
******************************************************************************)
METHOD PRIVATE addFailed : BOOL
VAR_INPUT
	bFatal : BOOL;
END_VAR

	u32Failed := u32Failed + 1;
	
	o_eResult := EResult_t.eStateFailed;
	
	IF bFatal = true THEN
		o_eResult := EResult_t.eStateFailedFatal;
		logError(concat('Test Failed Fatal: ', strId));
	ELSE
		logError(concat('Test Failed : ', strId));
	END_IF
END_METHOD

(******************************************************************************
Baustein: FB_UnitTestBase.addPassed
Spezifikation: doc/Spezifikation.pdf, Kap. x.y.z
-------------------------------------------------------------------------------
erstellt:
von:
Geändert:
von:
-------------------------------------------------------------------------------
Beschreibung
Diese Methode

-------------------------------------------------------------------------------
Input
-

Output
-
******************************************************************************)
METHOD PRIVATE addPassed : BOOL
VAR_INPUT
END_VAR

	u32Passed := u32Passed + 1;
END_METHOD

(******************************************************************************
Baustein: FB_UnitTestBase.assertEQUAL
Spezifikation: doc/Spezifikation.pdf, Kap. x.y.z
-------------------------------------------------------------------------------
erstellt:
von:
Geändert:
von:
-------------------------------------------------------------------------------
Beschreibung
Diese Methode

-------------------------------------------------------------------------------
Input
	Actual   : ANY;
	Expected : ANY;

Output
-
******************************************************************************)
METHOD PROTECTED assertEQUAL : BOOL
VAR_INPUT
	Actual   : ANY;
	Expected : ANY;
END_VAR

	assertEQUAL := FALSE;
	
	IF validate(Actual, Expected) = FALSE THEN
		addFailed(true);
		RETURN;
	END_IF
	
	assertTrue(MEMCMP(Actual.pValue, Expected.pValue, TO_UDINT(Actual.diSize)) = 0);
END_METHOD

(******************************************************************************
Baustein: FB_UnitTestBase.assertEQUAL_Fatal
Spezifikation: doc/Spezifikation.pdf, Kap. x.y.z
-------------------------------------------------------------------------------
erstellt:
von:
Geändert:
von:
-------------------------------------------------------------------------------
Beschreibung
Diese Methode

-------------------------------------------------------------------------------
Input
	Actual   : ANY;
	Expected : ANY;

Output
-
******************************************************************************)
METHOD PROTECTED assertEQUAL_Fatal : BOOL
VAR_INPUT
	Actual   : ANY;
	Expected : ANY;
END_VAR

	assertEQUAL_Fatal := FALSE;
	
	IF validate(Actual, Expected) = FALSE THEN
		addFailed(true);
		RETURN;
	END_IF

	assertTrue_Fatal(MEMCMP(Actual.pValue, Expected.pValue, TO_UDINT(Actual.diSize)) = 0);
END_METHOD

(******************************************************************************
Baustein: FB_UnitTestBase.assertFALSE
Spezifikation: doc/Spezifikation.pdf, Kap. x.y.z
-------------------------------------------------------------------------------
erstellt:
von:
Geändert:
von:
-------------------------------------------------------------------------------
Beschreibung
Diese Methode...

-------------------------------------------------------------------------------
Input
	bValue : BOOL;

Output
-
******************************************************************************)
METHOD PROTECTED assertFALSE : BOOL
VAR_INPUT
	bValue : BOOL;
END_VAR

	IF bValue = FALSE THEN
		addPassed();
	ELSE
		addFailed(bFatal := FALSE);
	END_IF
END_METHOD

(******************************************************************************
Baustein: FB_UnitTestBase.assertFALSE_Fatal
Spezifikation: doc/Spezifikation.pdf, Kap. x.y.z
-------------------------------------------------------------------------------
erstellt:
von:
Geändert:
von:
-------------------------------------------------------------------------------
Beschreibung
Diese Methode

-------------------------------------------------------------------------------
Input
	bValue : BOOL;

Output
-
******************************************************************************)
METHOD PROTECTED assertFALSE_Fatal : BOOL
VAR_INPUT
	bValue : BOOL;
END_VAR

	IF bValue = FALSE THEN
		addPassed();
	ELSE
		addFailed(bFatal := true);
	END_IF
END_METHOD

(******************************************************************************
Baustein: FB_UnitTestBase.assertNotEqual
Spezifikation: doc/Spezifikation.pdf, Kap. x.y.z
-------------------------------------------------------------------------------
erstellt:
von:
Geändert:
von:
-------------------------------------------------------------------------------
Beschreibung
Diese Methode

-------------------------------------------------------------------------------
Input
	Actual   : ANY;
	Expected : ANY;

Output
-
******************************************************************************)
METHOD PROTECTED assertNotEqual : BOOL
VAR_INPUT
	Actual   : ANY;
	Expected : ANY;
END_VAR

	assertNotEqual := FALSE;
	
	IF validate(Actual, Expected) = FALSE THEN
		addFailed(true);
		RETURN;
	END_IF
	
	assertTrue(MEMCMP(Actual.pValue, Expected.pValue, TO_UDINT(Actual.diSize)) <> 0);
END_METHOD

(******************************************************************************
Baustein: FB_UnitTestBase.assertNotEqual_Fatal
Spezifikation: doc/Spezifikation.pdf, Kap. x.y.z
-------------------------------------------------------------------------------
erstellt:
von:
Geändert:
von:
-------------------------------------------------------------------------------
Beschreibung
Diese Methode

-------------------------------------------------------------------------------
Input
	Actual   : ANY;
	Expected : ANY;

Output
-
******************************************************************************)
METHOD PROTECTED assertNotEqual_Fatal : BOOL
VAR_INPUT
	Actual   : ANY;
	Expected : ANY;
END_VAR

	assertNotEqual_Fatal := FALSE;
	
	IF validate(Actual, Expected) = FALSE THEN
		addFailed(true);
		RETURN;
	END_IF
	
	assertTrue_Fatal(MEMCMP(Actual.pValue, Expected.pValue, TO_UDINT(Actual.diSize)) <> 0);
END_METHOD

(******************************************************************************
Baustein: FB_UnitTestBase.assertPtrEqual
Spezifikation: doc/Spezifikation.pdf, Kap. x.y.z
-------------------------------------------------------------------------------
erstellt:
von:
Geändert:
von:
-------------------------------------------------------------------------------
Beschreibung
Diese Methode

-------------------------------------------------------------------------------
Input
	pActual   : PVOID;
	pExpected : PVOID;
	
Output
-
******************************************************************************)
METHOD PROTECTED assertPtrEqual : BOOL
VAR_INPUT
	pActual   : PVOID;
	pExpected : PVOID;
END_VAR

	assertTRUE(pActual = pExpected);
END_METHOD

(******************************************************************************
Baustein: FB_UnitTestBase.assertPtrEqual_Fatal
Spezifikation: doc/Spezifikation.pdf, Kap. x.y.z
-------------------------------------------------------------------------------
erstellt:
von:
Geändert:
von:
-------------------------------------------------------------------------------
Beschreibung
Diese Methode

-------------------------------------------------------------------------------
Input
	pActual   : PVOID;
	pExpected : PVOID;

Output
-
******************************************************************************)
METHOD PROTECTED assertPtrEqual_Fatal : BOOL
VAR_INPUT
	pActual   : PVOID;
	pExpected : PVOID;
END_VAR

	assertTRUE_Fatal(pActual = pExpected);
END_METHOD

(******************************************************************************
Baustein: FB_UnitTestBase.assertPtrNotEqual
Spezifikation: doc/Spezifikation.pdf, Kap. x.y.z
-------------------------------------------------------------------------------
erstellt:
von:
Geändert:
von:
-------------------------------------------------------------------------------
Beschreibung
Diese Methode

-------------------------------------------------------------------------------
Input
	pActual   : PVOID;
	pExpected : PVOID;

Output
-
******************************************************************************)
METHOD PROTECTED assertPtrNotEqual : BOOL
VAR_INPUT
	pActual   : PVOID;
	pExpected : PVOID;
END_VAR

	assertTRUE(pActual <> pExpected);
END_METHOD

(******************************************************************************
Baustein: FB_UnitTestBase.assertPtrNotEqual_Fatal
Spezifikation: doc/Spezifikation.pdf, Kap. x.y.z
-------------------------------------------------------------------------------
erstellt:
von:
Geändert:
von:
-------------------------------------------------------------------------------
Beschreibung
Diese Methode

-------------------------------------------------------------------------------
Input
	pActual   : PVOID;
	pExpected : PVOID;

Output
-
******************************************************************************)
METHOD PROTECTED assertPtrNotEqual_Fatal : BOOL
VAR_INPUT
	pActual   : PVOID;
	pExpected : PVOID;
END_VAR

	assertTRUE_Fatal(pActual <> pExpected);
END_METHOD

(******************************************************************************
Baustein: FB_UnitTestBase.assertPtrNotNull
Spezifikation: doc/Spezifikation.pdf, Kap. x.y.z
-------------------------------------------------------------------------------
erstellt:
von:
Geändert:
von:
-------------------------------------------------------------------------------
Beschreibung
Diese Methode

-------------------------------------------------------------------------------
Input
	pActual   : PVOID;

Output
-
******************************************************************************)
METHOD PROTECTED assertPtrNotNull : BOOL
VAR_INPUT
	pActual   : PVOID;
END_VAR

	assertTRUE(pActual <> 0);
END_METHOD

(******************************************************************************
Baustein: FB_UnitTestBase.assertPtrNotNull_Fatal
Spezifikation: doc/Spezifikation.pdf, Kap. x.y.z
-------------------------------------------------------------------------------
erstellt:
von:
Geändert:
von:
-------------------------------------------------------------------------------
Beschreibung
Diese Methode

-------------------------------------------------------------------------------
Input
	pActual   : PVOID;

Output
-
******************************************************************************)
METHOD PROTECTED assertPtrNotNull_Fatal : BOOL
VAR_INPUT
	pActual   : PVOID;
END_VAR

	assertTRUE_Fatal(pActual <> 0);
END_METHOD

(******************************************************************************
Baustein: FB_UnitTestBase.assertPtrNull
Spezifikation: doc/Spezifikation.pdf, Kap. x.y.z
-------------------------------------------------------------------------------
erstellt:
von:
Geändert:
von:
-------------------------------------------------------------------------------
Beschreibung
Diese Methode

-------------------------------------------------------------------------------
Input
	pActual   : PVOID;

Output
-
******************************************************************************)
METHOD PROTECTED assertPtrNull : BOOL
VAR_INPUT
	pActual   : PVOID;
END_VAR

	assertTRUE(pActual = 0);
END_METHOD

(******************************************************************************
Baustein: FB_UnitTestBase.assertPtrNull_Fatal
Spezifikation: doc/Spezifikation.pdf, Kap. x.y.z
-------------------------------------------------------------------------------
erstellt:
von:
Geändert:
von:
-------------------------------------------------------------------------------
Beschreibung
Diese Methode

-------------------------------------------------------------------------------
Input
	pActual   : PVOID;

Output
-
******************************************************************************)
METHOD PROTECTED assertPtrNull_Fatal : BOOL
VAR_INPUT
	pActual   : PVOID;
END_VAR

	assertTRUE_Fatal(pActual = 0);
END_METHOD

(******************************************************************************
Baustein: FB_UnitTestBase.assertRealEqual
Spezifikation: doc/Spezifikation.pdf, Kap. x.y.z
-------------------------------------------------------------------------------
erstellt:
von:
Geändert:
von:
-------------------------------------------------------------------------------
Beschreibung
Diese Methode

-------------------------------------------------------------------------------
Input
	r32Actual 		: REAL;
	r32Expected 	: REAL;
	r32Granularity 	: REAL;

Output
-
******************************************************************************)
METHOD PROTECTED assertRealEqual : BOOL
VAR_INPUT
	r32Actual 		: REAL;
	r32Expected 	: REAL;
	r32Granularity 	: REAL;
END_VAR

	assertTRUE(ABS(r32Actual-r32Expected) <= ABS(r32Granularity));
END_METHOD

(******************************************************************************
Baustein: FB_UnitTestBase.assertRealEqual_Fatal
Spezifikation: doc/Spezifikation.pdf, Kap. x.y.z
-------------------------------------------------------------------------------
erstellt:
von:
Geändert:
von:
-------------------------------------------------------------------------------
Beschreibung
Diese Methode

-------------------------------------------------------------------------------
Input
	r32Actual 		: REAL;
	r32Expected 	: REAL;
	r32Granularity 	: REAL;

Output
-
******************************************************************************)
METHOD PROTECTED assertRealEqual_Fatal : BOOL
VAR_INPUT
	r32Actual 		: REAL;
	r32Expected 	: REAL;
	r32Granularity 	: REAL;
END_VAR

	assertTRUE_Fatal(ABS(r32Actual-r32Expected) <= ABS(r32Granularity));
END_METHOD

(******************************************************************************
Baustein: FB_UnitTestBase.assertRealNotEqual
Spezifikation: doc/Spezifikation.pdf, Kap. x.y.z
-------------------------------------------------------------------------------
erstellt:
von:
Geändert:
von:
-------------------------------------------------------------------------------
Beschreibung
Diese Methode

-------------------------------------------------------------------------------
Input
	r32Actual 		: REAL;
	r32Expected 	: REAL;
	r32Granularity 	: REAL;

Output
-
******************************************************************************)
METHOD PRIVATE assertRealNotEqual : BOOL
VAR_INPUT
	r32Actual 		: REAL;
	r32Expected 	: REAL;
	r32Granularity 	: REAL;
END_VAR

	assertTRUE(ABS(r32Actual-r32Expected) > ABS(r32Granularity));
END_METHOD

(******************************************************************************
Baustein: FB_UnitTestBase.assertRealNotEqual_Fatal
Spezifikation: doc/Spezifikation.pdf, Kap. x.y.z
-------------------------------------------------------------------------------
erstellt:
von:
Geändert:
von:
-------------------------------------------------------------------------------
Beschreibung
Diese Methode

-------------------------------------------------------------------------------
Input
	r32Actual 		: REAL;
	r32Expected 	: REAL;
	r32Granularity 	: REAL;

Output
-
******************************************************************************)
METHOD PROTECTED assertRealNotEqual_Fatal : BOOL
VAR_INPUT
	r32Actual 		: REAL;
	r32Expected 	: REAL;
	r32Granularity 	: REAL;
END_VAR

	assertTRUE_Fatal(ABS(r32Actual-r32Expected) > ABS(r32Granularity));
END_METHOD

(******************************************************************************
Baustein: FB_UnitTestBase.assertStringEqual
Spezifikation: doc/Spezifikation.pdf, Kap. x.y.z
-------------------------------------------------------------------------------
erstellt:
von:
Geändert:
von:
-------------------------------------------------------------------------------
Beschreibung
Diese Methode

-------------------------------------------------------------------------------
Input
	pActual 	: StringHandle_t;
	pExpected 	: StringHandle_t;

Output
-
******************************************************************************)
METHOD PROTECTED assertStringEqual : BOOL
VAR_INPUT
	pActual 	: StringHandle_t;
	pExpected 	: StringHandle_t;
END_VAR

	IF strncmp(pActual, pExpected, LEN(pExpected^)) = TRUE THEN
		addPassed();
	ELSE
		addFailed(bFatal := FALSE);		
	END_IF
END_METHOD

(******************************************************************************
Baustein: FB_UnitTestBase.assertStringEqual_Fatal
Spezifikation: doc/Spezifikation.pdf, Kap. x.y.z
-------------------------------------------------------------------------------
erstellt:
von:
Geändert:
von:
-------------------------------------------------------------------------------
Beschreibung
Diese Methode

-------------------------------------------------------------------------------
Input
	pActual 	: StringHandle_t;
	pExpected 	: StringHandle_t;

Output
-
******************************************************************************)
METHOD PROTECTED assertStringEqual_Fatal : BOOL
VAR_INPUT
	pActual 	: StringHandle_t;
	pExpected 	: StringHandle_t;
END_VAR

	IF strncmp(pActual, pExpected, LEN(pExpected^)) = TRUE THEN
		addPassed();
	ELSE
		addFailed(bFatal := TRUE);		
	END_IF
END_METHOD

(******************************************************************************
Baustein: FB_UnitTestBase.assertStringNotEqual
Spezifikation: doc/Spezifikation.pdf, Kap. x.y.z
-------------------------------------------------------------------------------
erstellt:
von:
Geändert:
von:
-------------------------------------------------------------------------------
Beschreibung
Diese Methode

-------------------------------------------------------------------------------
Input
	pActual 	: StringHandle_t;
	pExpected 	: StringHandle_t;

Output
-
******************************************************************************)
METHOD PROTECTED assertStringNotEqual : BOOL
VAR_INPUT
	pActual 	: StringHandle_t;
	pExpected 	: StringHandle_t;
END_VAR

	IF strncmp(pActual, pExpected, LEN(pExpected^)) = false THEN
		addPassed();
	ELSE
		addFailed(bFatal := FALSE);		
	END_IF
END_METHOD

(******************************************************************************
Baustein: FB_UnitTestBase.assertStringNotEqual_fatal
Spezifikation: doc/Spezifikation.pdf, Kap. x.y.z
-------------------------------------------------------------------------------
erstellt:
von:
Geändert:
von:
-------------------------------------------------------------------------------
Beschreibung
Diese Methode

-------------------------------------------------------------------------------
Input
	pExpected 	: StringHandle_t;
	pActual 	: StringHandle_t;

Output
-
******************************************************************************)
METHOD PROTECTED assertStringNotEqual_fatal : BOOL
VAR_INPUT
	pExpected 	: StringHandle_t;
	pActual 	: StringHandle_t;
END_VAR

	IF strncmp(pActual, pExpected, LEN(pExpected^)) = FALSE THEN
		addPassed();
	ELSE
		addFailed(bFatal := TRUE);		
	END_IF
END_METHOD

(******************************************************************************
Baustein: FB_UnitTestBase.assertTRUE
Spezifikation: doc/Spezifikation.pdf, Kap. x.y.z
-------------------------------------------------------------------------------
erstellt:
von:
Geändert:
von:
-------------------------------------------------------------------------------
Beschreibung
Diese Methode...

-------------------------------------------------------------------------------
Input
	bValue : BOOL;

Output
-
******************************************************************************)
METHOD PROTECTED assertTRUE : BOOL
VAR_INPUT
	bValue : BOOL;
END_VAR

	IF bValue = true THEN
		addPassed();
	ELSE
		addFailed(bFatal := FALSE);
	END_IF
END_METHOD


(******************************************************************************
Baustein: FB_UnitTestBase.assertTRUE_Fatal
Spezifikation: doc/Spezifikation.pdf, Kap. x.y.z
-------------------------------------------------------------------------------
erstellt:
von:
Geändert:
von:
-------------------------------------------------------------------------------
Beschreibung
Diese Methode

-------------------------------------------------------------------------------
Input
-

Output
-
******************************************************************************)
METHOD PROTECTED assertTRUE_Fatal : BOOL
VAR_INPUT
	bValue : BOOL;
END_VAR

	IF bValue = TRUE THEN
		addPassed();
	ELSE
		addFailed(bFatal := true);
	END_IF
END_METHOD

(******************************************************************************
Baustein: FB_UnitTestBase.cleanup
Spezifikation: doc/Spezifikation.pdf, Kap. x.y.z
-------------------------------------------------------------------------------
erstellt:
von:
Geändert:
von:
-------------------------------------------------------------------------------
Beschreibung
Diese Methode...

-------------------------------------------------------------------------------
Input
-

Output
-
******************************************************************************)
METHOD PUBLIC cleanup : BOOL
VAR_INPUT
END_VAR

	cleanup := TRUE;
END_METHOD

(******************************************************************************
Baustein: FB_UnitTestBase.execute
Spezifikation: doc/Spezifikation.pdf, Kap. x.y.z
-------------------------------------------------------------------------------
erstellt:
von:
Geändert:
von:
-------------------------------------------------------------------------------
Beschreibung
Diese Methode...

-------------------------------------------------------------------------------
Input
-

Output
-
******************************************************************************)
METHOD PUBLIC execute : BOOL
VAR_INPUT
END_VAR

	Execute := TRUE;
END_METHOD

(******************************************************************************
Baustein: FB_Testsuite.FB_init
Spezifikation: doc/Spezifikation.pdf, Kap. x.y.z
-------------------------------------------------------------------------------
erstellt:
von:
Geändert:
von:
-------------------------------------------------------------------------------
Beschreibung
Diese Methode

-------------------------------------------------------------------------------
Input
-

Output
-
******************************************************************************)
METHOD FB_init : BOOL
VAR_INPUT
	bInitRetains 	: BOOL; // if TRUE, the retain variables are initialized (warm start / cold start)
	bInCopyCode 	: BOOL;  // if TRUE, the instance afterwards gets moved into the copy code (online change)
	i_strId	  		: ObjectId_t;
	i_pTestSuite 	: TestSuiteHandle_t;
	i_bExecute      : BOOL := true; 
END_VAR
	
	strId 		:= i_strId;
	pTestSuite 	:= i_pTestSuite;
	
	register();
END_METHOD

(******************************************************************************
Baustein: FB_UnitTestBase.getFailed
Spezifikation: doc/Spezifikation.pdf, Kap. x.y.z
-------------------------------------------------------------------------------
erstellt:
von:
Geändert:
von:
-------------------------------------------------------------------------------
Beschreibung
Diese Methode

-------------------------------------------------------------------------------
Input
-

Output
-
******************************************************************************)
METHOD PUBLIC getFailed : UDINT
VAR_INPUT
END_VAR

	getFailed := u32Failed;
END_METHOD

(******************************************************************************
Baustein: FB_UnitTestBase.getPassed
Spezifikation: doc/Spezifikation.pdf, Kap. x.y.z
-------------------------------------------------------------------------------
erstellt:
von:
Geändert:
von:
-------------------------------------------------------------------------------
Beschreibung
Diese Methode

-------------------------------------------------------------------------------
Input
-

Output
-
******************************************************************************)
METHOD PUBLIC getPassed : UDINT
VAR_INPUT
END_VAR

	getPassed := u32Passed;
END_METHOD

(******************************************************************************
Baustein: FB_UnitTestBase.logError
Spezifikation: doc/Spezifikation.pdf, Kap. x.y.z
-------------------------------------------------------------------------------
erstellt:
von:
Geändert:
von:
-------------------------------------------------------------------------------
Beschreibung
Diese Methode

-------------------------------------------------------------------------------
Input
-

Output
-
******************************************************************************)
METHOD PROTECTED logError : BOOL
VAR_INPUT
	i_strMessage : StrMessage_t;
END_VAR

	ADSLOGSTR(msgCtrlMask 	:= ADSLOG_MSGTYPE_ERROR , 
			  msgFmtStr 	:= i_strMessage, 
			  strArg 		:= '');
END_METHOD

(******************************************************************************
Baustein: FB_UnitTestBase.logInfo
Spezifikation: doc/Spezifikation.pdf, Kap. x.y.z
-------------------------------------------------------------------------------
erstellt:
von:
Geändert:
von:
-------------------------------------------------------------------------------
Beschreibung
Diese Methode

-------------------------------------------------------------------------------
Input
-

Output
-
******************************************************************************)
METHOD PROTECTED logInfo : BOOL
VAR_INPUT
	i_strMessage : StrMessage_t;
END_VAR

	ADSLOGSTR(msgCtrlMask 	:= ADSLOG_MSGTYPE_HINT , 
			  msgFmtStr 	:= i_strMessage, 
			  strArg 		:= '');
END_METHOD

(******************************************************************************
Baustein: FB_UnitTestBase.prepare
Spezifikation: doc/Spezifikation.pdf, Kap. x.y.z
-------------------------------------------------------------------------------
erstellt:
von:
Geändert:
von:
-------------------------------------------------------------------------------
Beschreibung
Diese Methode...

-------------------------------------------------------------------------------
Input
-

Output
-
******************************************************************************)
METHOD PUBLIC prepare : BOOL
VAR_INPUT
END_VAR

	u32Passed := 0;
	u32Failed := 0;
	
	prepare := true;
END_METHOD

(******************************************************************************
Baustein: FB_UnitTestBase.register
Spezifikation: doc/Spezifikation.pdf, Kap. x.y.z
-------------------------------------------------------------------------------
erstellt:
von:
Geändert:
von:
-------------------------------------------------------------------------------
Beschreibung
Diese Methode

-------------------------------------------------------------------------------
Input
-

Output
-
******************************************************************************)
METHOD PROTECTED register : BOOL
VAR_INPUT
END_VAR

	IF pTestSuite <> 0 	AND 
       bRegistered = FALSE  THEN
		
		bRegistered := pTestSuite^.addTestcase(THIS);
	
	END_IF
END_METHOD

(******************************************************************************
Baustein: FB_UnitTestBase.strncmp
Spezifikation: doc/Spezifikation.pdf, Kap. x.y.z
-------------------------------------------------------------------------------
erstellt:
von:
Geändert:
von:
-------------------------------------------------------------------------------
Beschreibung
Diese Methode

-------------------------------------------------------------------------------
Input
	strInput 	: StringHandle_t;
	strCompare 	: StringHandle_t;
	s16Size		: INT;

Output
-
******************************************************************************)
METHOD PRIVATE strncmp : BOOL
VAR_INPUT
	strInput 	: StringHandle_t;
	strCompare 	: StringHandle_t;
	s16Size		: INT;
END_VAR
VAR
	s16Size1 : INT;
	s16Size2 : INT;
	s16Diff  : INT;
END_VAR

   s16Size1:= LEN(strInput^); 
	s16Size2:= LEN(strCompare^); 
	
	strncmp := FALSE;
	
	s16Diff := s16Size1 - s16Size2;
   
	// vergleich nur wenn beide Strings
	// gleich groß sind.
	IF s16Diff  = 0 THEN

		strncmp := TRUE;
	
		WHILE(s16Size > 0) DO

			IF strInput^ <> strCompare^ THEN
				strncmp := FALSE;
			END_IF;  
 
			strInput   := strInput + 1;
			strCompare := strCompare + 1;
			s16Size    := s16Size - 1;

		END_WHILE


	
	END_IF;
END_METHOD

(******************************************************************************
Baustein: FB_UnitTestBase.validate
Spezifikation: doc/Spezifikation.pdf, Kap. x.y.z
-------------------------------------------------------------------------------
erstellt:
von:
Geändert:
von:
-------------------------------------------------------------------------------
Beschreibung
Diese Methode

-------------------------------------------------------------------------------
Input
	var1 : ANY;
	var2 : ANY;

Output
-
******************************************************************************)
METHOD PRIVATE validate : BOOL
VAR_INPUT
	var1 : ANY;
	var2 : ANY;
END_VAR

	validate := FALSE;
	
	IF (var1.pValue = 0 OR var2.pValue = 0) THEN
		RETURN;
	END_IF

	IF (var1.TypeClass <> var2.TypeClass) THEN
		RETURN;
	END_IF;	
	
	IF (var1.diSize <> var2.diSize) THEN
		RETURN;
	END_IF;	
	
	validate := true;
END_METHOD

END_FUNCTION_BLOCK

// ---- Source/Report/FB_FileBase.TcPOU
(******************************************************************************
Baustein: FB_TestReportBase
Spezifikation: doc/Spezifikation.pdf, Kap. x.y.z
-------------------------------------------------------------------------------
erstellt:
von:
Geändert:
von:
-------------------------------------------------------------------------------
Beschreibung
Dieser Baustein enthält alle zugeordneten Testfälle. Ein Testfall
ist ein abgeleiteter Baustein (FB) von FB_UnitTestBase.

-------------------------------------------------------------------------------
Input
-

Output
-
******************************************************************************)
FUNCTION_BLOCK FB_FileBase
VAR_INPUT
END_VAR
VAR_OUTPUT
	o_bOpen 	: BOOL;
	o_bError 	: BOOL;
	o_bEmpty 	: BOOL;
END_VAR
VAR
	Buffer      : ARRAY[0..1024] OF BYTE;
	u32RdIdx    : UDINT;
	u32WrIdx    : UDINT;
	u32MaxIdx   : UDINT := 1024;
	
	fbOpen      : FB_FileOpen;
	fbClose     : FB_FileClose;
	fbWrite	    : FB_FileWrite;
	strFileName : StrFileName_t;
	strFilePath : StrPathName_t;
	
	eState 		: EExportState_t;
	u32Line     : UDINT;
	
	sStatistic  : SStatistic_t;

	trgOpen 	: F_TRIG;
	trgWrite 	: F_TRIG;
	trgClose 	: F_TRIG;
END_VAR


	fbOpen();
	fbWrite();
	fbClose();
	
	trgOpen(CLK := fbOpen.bBusy);
	IF trgOpen.Q = TRUE THEN
		fbOpen.bExecute := FALSE;
	END_IF;

	trgWrite(CLK := fbWrite.bBusy);
	IF trgWrite.Q = TRUE THEN
		fbWrite.bExecute := FALSE;
	END_IF;

	trgClose(CLK := fbClose.bBusy);
	IF trgClose.Q = TRUE THEN
		fbClose.bExecute := FALSE;
	END_IF;

	o_bEmpty := (u32WrIdx = u32RdIdx);

(******************************************************************************
Baustein: FB_TestReportBase.addCrlf
Spezifikation: doc/Spezifikation.pdf, Kap. x.y.z
-------------------------------------------------------------------------------
erstellt:
von:
Geändert:
von:
-------------------------------------------------------------------------------
Beschreibung


-------------------------------------------------------------------------------
Input
-

Output
-
******************************************************************************)
METHOD PUBLIC addCrlf : ERetCode_t
VAR_INPUT
END_VAR
VAR
	strTemp : string := '$R$N';
END_VAR

	addData(adr(strTemp), 2);
	
	addCrlf := ERetCode_t.eRetDone;
END_METHOD

METHOD PRIVATE addData : BOOL
VAR_INPUT
	pData   : POINTER TO BYTE;
	u32Size : UDINT;
END_VAR
VAR
	u32Part1 : UDINT;
	u32Part2 : UDINT;
END_VAR

	IF u32WrIdx + u32Size <= u32MaxIdx THEN
		MemCpy(ADR(buffer)+u32WrIdx, pData, u32Size);
		u32WrIdx := u32WrIdx + u32Size;
	ELSE
		// buffer bis maximum beschreiben und den rest
		// vorne einfügen
		u32Part1 := u32MaxIdx-u32WrIdx;
		u32Part2 := u32Size - u32Part1;

		MemCpy(ADR(buffer) + u32WrIdx, pData, u32Part1);
		
		MemCpy(ADR(buffer), pData+u32Part1, u32Part2);
		// Schreibindex ist dann die Restgröße in Byte
		u32WrIdx := u32Part2;
	END_IF
END_METHOD

(******************************************************************************
Baustein: FB_TestReportBase.addString
Spezifikation: doc/Spezifikation.pdf, Kap. x.y.z
-------------------------------------------------------------------------------
erstellt:
von:
Geändert:
von:
-------------------------------------------------------------------------------
Beschreibung

-------------------------------------------------------------------------------
Input
	i_strData : STRING(255);

Output
-
******************************************************************************)
METHOD PUBLIC addString : ERetCode_t
VAR_INPUT
	i_strData : STRING(255);
END_VAR

	addData(ADR(i_strData), len(i_strData));
	
	addString := ERetcode_t.eRetDone;
END_METHOD

(******************************************************************************
Baustein: FB_TestReportBase.addValue
Spezifikation: doc/Spezifikation.pdf, Kap. x.y.z
-------------------------------------------------------------------------------
erstellt:
von:
Geändert:
von:
-------------------------------------------------------------------------------
Beschreibung

-------------------------------------------------------------------------------
Input
	i_anyValue : ANY;

Output
-
******************************************************************************)
METHOD PUBLIC addValue : ERetCode_t
VAR_INPUT
	i_anyValue : ANY;
END_VAR
VAR
	uValue : UBaseTypes_t;
END_VAR

	addValue  := ERetcode_t.eRetDone;
	
	IF i_anyValue.pValue = 0 THEN
		addValue  := ERetcode_t.eRetFailed;
		RETURN;
	END_IF

	MEMCPY(ADR(uValue),i_anyValue.pValue, TO_UDINT(i_anyValue.diSize)); 

	CASE i_anyValue.TypeClass OF

	IBaseLibrary.TYPE_SINT:

		addString(SINT_TO_STRING(uValue.s8Value));

	IBaseLibrary.TYPE_USINT:

		addString(USINT_TO_STRING(uValue.u8Value));

	IBaseLibrary.TYPE_INT:

		addString(INT_TO_STRING(uValue.s16Value));

	IBaseLibrary.TYPE_DINT:

		addString(DINT_TO_STRING(uValue.s32Value));

	IBaseLibrary.TYPE_UINT:

		addString(UINT_TO_STRING(uValue.u16Value));

	IBaseLibrary.TYPE_UDINT:

		addString(UDINT_TO_STRING(uValue.u32Value));

	IBaseLibrary.TYPE_WORD:

		addString(WORD_TO_STRING(uValue.w16Value));

	IBaseLibrary.TYPE_DWORD:

		addString(DWORD_TO_STRING(uValue.w32Value));

	IBaseLibrary.TYPE_BYTE:

		addString(BYTE_TO_STRING(uValue.u8Value));

	IBaseLibrary.TYPE_BOOL:
		
		IF (uValue.bValue = TRUE) THEN
			addString('TRUE');
		ELSE
			addString('FALSE');
		END_IF;

	IBaseLibrary.TYPE_REAL:
		
		addString(REAL_TO_STRING(uValue.r32Value));
	
	ELSE
		ADSLOGSTR(msgCtrlMask 	:= ADSLOG_MSGTYPE_ERROR , 
				  msgFmtStr 	:= 'TestReportBase.AddValue: Unbekannter Datentyp!', 
				  strArg 		:= '');
	END_CASE;
END_METHOD

(******************************************************************************
Baustein: FB_TestReportBase.clearBuffer
Spezifikation: doc/Spezifikation.pdf, Kap. x.y.z
-------------------------------------------------------------------------------
erstellt:
von:
Geändert:
von:
-------------------------------------------------------------------------------
Beschreibung

-------------------------------------------------------------------------------
Input
-

Output
-
******************************************************************************)
METHOD PUBLIC clearBuffer : ERetCode_t
VAR_INPUT
END_VAR

	clearBuffer := ERetCode_t.eRetDone;
	
	MemSet(ADR(buffer), 0, SIZEOF(buffer));
	
	u32WrIdx := u32RdIdx := 0;
END_METHOD

(******************************************************************************
Baustein: FB_TestReportBase.Close
Spezifikation: doc/Spezifikation.pdf, Kap. x.y.z
-------------------------------------------------------------------------------
erstellt:
von:
Geändert:
von:
-------------------------------------------------------------------------------
Beschreibung


-------------------------------------------------------------------------------
Input
-

Output
-
******************************************************************************)
METHOD PUBLIC Close : ERetCode_t
VAR_INPUT
END_VAR

	Close := ERetCode_t.eRetFailed;
	
	fbClose.hFile 		:= fbOpen.hFile;

	IF o_bEmpty = TRUE THEN

		fbClose.bExecute 	:= TRUE; 

		IF trgClose.Q = TRUE THEN
			o_bOpen 			:= FALSE;
			Close 				:= ERetCode_t.eRetDone;
			fbClose.bExecute 	:= FALSE;		
		ELSE	
			Close := ERetCode_t.eRetBusy;
		END_IF;	
		
		IF fbClose.bError = TRUE THEN
			Close := eRetCode_t.eRetFailed;
		END_IF;			

	ELSE
		Close := ERetCode_t.eRetBusy;
	END_IF;
END_METHOD

(******************************************************************************
Baustein: FB_TestReportBase.getFileName
Spezifikation: doc/Spezifikation.pdf, Kap. x.y.z
-------------------------------------------------------------------------------
erstellt:
von:
Geändert:
von:
-------------------------------------------------------------------------------
Beschreibung
Diese Methode muss vom ableitenden Baustein überschrieben werden und
wird von der Basisklasse aus aufgerufen wenn der Report erstellt werden
soll.

-------------------------------------------------------------------------------
Input
	i_pFileName : NameHandle_t;
	i_pPath		: PathHandle_t;

Output
-
******************************************************************************)
METHOD PROTECTED getFileName : ERetCode_t
VAR_INPUT
	i_pFileName : NameHandle_t;
	i_pPath		: PathHandle_t;
END_VAR
END_METHOD

(******************************************************************************
Baustein: FB_TestReportBase.getTime
Spezifikation: doc/Spezifikation.pdf, Kap. x.y.z
-------------------------------------------------------------------------------
erstellt:
von:
Geändert:
von:
-------------------------------------------------------------------------------
Beschreibung


-------------------------------------------------------------------------------
Input
-

Output
-
******************************************************************************)
METHOD PROTECTED getTime : TimeStruct
VAR_INPUT
END_VAR
VAR
END_VAR

	getTime := PRG_UnitTestLib.getTime();
END_METHOD

(******************************************************************************
Baustein: FB_TestReportBase.Open
Spezifikation: doc/Spezifikation.pdf, Kap. x.y.z
-------------------------------------------------------------------------------
erstellt:
von:
Geändert:
von:
-------------------------------------------------------------------------------
Beschreibung


-------------------------------------------------------------------------------
Input
-

Output
-
******************************************************************************)
METHOD PUBLIC open : ERetCode_t
VAR_INPUT
	i_strPath : StrPathName_t;
	i_strName : StrFileName_t;
END_VAR

	open := ERetCode_t.eRetFailed;
	
	strFileName := i_strName;
	strFilePath := i_strPath;

	fbOpen.sPathName := CONCAT(strFilePath, strFileName);
	fbOpen.nMode 	 := FOPEN_MODEWRITE OR FOPEN_MODEBINARY;	
	fbOpen.bExecute  := TRUE;
			
	IF trgOpen.Q = TRUE THEN
		o_bOpen := true;
		open := ERetCode_t.eRetDone;
		fbOpen.bExecute  := FALSE;		
	ELSE	
		open := ERetCode_t.eRetBusy;
	END_IF;	
	
	IF fbOpen.bError = TRUE THEN
		open := eRetCode_t.eRetFailed;
	END_IF;
END_METHOD

(******************************************************************************
Baustein: FB_TestReportBase.reset
Spezifikation: doc/Spezifikation.pdf, Kap. x.y.z
-------------------------------------------------------------------------------
erstellt:
von:
Geändert:
von:
-------------------------------------------------------------------------------
Beschreibung


-------------------------------------------------------------------------------
Input
-

Output
-
******************************************************************************)
METHOD PUBLIC reset : BOOL
VAR_INPUT
END_VAR

	IF fbOpen.hFile <> 0 THEN
		close();
	END_IF
	
	clearBuffer();

	fbOpen(sPathName := '', bExecute := FALSE);
	
	fbWrite(bExecute := FALSE);
	
	fbClose(bExecute := FALSE);
	
	o_bOpen := false;
END_METHOD

(******************************************************************************
Baustein: FB_TestReportBase.writeBuffer
Spezifikation: doc/Spezifikation.pdf, Kap. x.y.z
-------------------------------------------------------------------------------
erstellt:
von:
Geändert:
von:
-------------------------------------------------------------------------------
Beschreibung


-------------------------------------------------------------------------------
Input
-

Output
-
******************************************************************************)
METHOD PUBLIC writeBuffer : ERetCode_t
VAR_INPUT
END_VAR
VAR
	u32Len : UDINT;
END_VAR

	writeBuffer := eRetCode_t.eRetBusy;

	IF fbWrite.bBusy = TRUE THEN
		RETURN;	
	ELSIF u32WrIdx = u32RdIdx THEN
		writeBuffer := eRetCode_t.eRetDone;
		RETURN;	
	END_IF
	
	IF u32WrIdx > u32RdIdx THEN
		u32Len := u32WrIdx - u32RdIdx; 
		writeBuffer := writeData(i_pData := ADR(Buffer)+u32RdIdx, u32Size := u32Len);	
	ELSE
		u32Len := u32MaxIdx - u32RdIdx; 
		writeBuffer := writeData(i_pData := ADR(Buffer)+ u32RdIdx, u32Size := u32Len);
		writeBuffer := writeData(i_pData := ADR(Buffer), u32Size := u32WrIdx);	
	END_IF;
END_METHOD

(******************************************************************************
Baustein: FB_TestReportBase.writeData
Spezifikation: doc/Spezifikation.pdf, Kap. x.y.z
-------------------------------------------------------------------------------
erstellt:
von:
Geändert:
von:
-------------------------------------------------------------------------------
Beschreibung


-------------------------------------------------------------------------------
Input
	i_pData : POINTER TO BYTE;
	u32Size : UDINT;
	
Output
-
******************************************************************************)
METHOD PROTECTED writeData : ERetCode_t
VAR_INPUT
	i_pData : POINTER TO BYTE;
	u32Size : UDINT;
END_VAR

	writeData := ERetCode_t.eRetFailed;
	
	IF u32Size = 0 OR i_pData = 0 THEN
		RETURN;
	END_IF
	
	fbWrite.pWriteBuff 	:= i_pData; 
	fbWrite.cbWriteLen 	:= u32Size; 
	fbWrite.hFile 		:= fbOpen.hFile; 

	fbWrite(bExecute 	:= TRUE);
			
	IF fbWrite.bBusy = FALSE THEN
		fbWrite(bExecute 	:= FALSE);	
		writeData 	:= ERetCode_t.eRetDone;
		u32RdIdx 	:= u32WrIdx;
	ELSE	
		writeData := ERetCode_t.eRetBusy;
	END_IF;	

	IF fbWrite.bError = TRUE THEN
		writeData := eRetCode_t.eRetFailed;
	END_IF;
END_METHOD

END_FUNCTION_BLOCK

// ---- Source/Report/FB_TextReport.TcPOU
FUNCTION_BLOCK FB_TextReport EXTENDS FB_TestReportBase
VAR_INPUT
END_VAR
VAR_OUTPUT
END_VAR
VAR
END_VAR

(******************************************************************************
Baustein: FB_TestReportBase.BuildFile
Spezifikation: doc/Spezifikation.pdf, Kap. x.y.z
-------------------------------------------------------------------------------
erstellt:
von:
Geändert:
von:
-------------------------------------------------------------------------------
Beschreibung
Diese Methode muss vom ableitenden Baustein überschrieben werden und
wird von der Basisklasse aus aufgerufen wenn der Report erstellt werden
soll.

-------------------------------------------------------------------------------
Input
-

Output
-
******************************************************************************)
METHOD PROTECTED BuildFile : ERetCode_t
VAR_INPUT
	i_u32Line : UDINT;
END_VAR

	BuildFile := ERetCode_t.eRetBusy;

	CASE i_u32Line OF

	0: addString('Test Report :');
	   addDate(getTime());
	   addString(' - ');
	   addTime(getTime());
	1: addString('++++++++++++++++++++++++++++++++++++++++++++++++++');
	2: //
	3: //

	4: addString('Asserts gesamt: ');
	   addValue(sStatistic.u32Asserts);

	5: addString('Asserts passed: ');
	   addValue(sStatistic.u32Passed);

	6: addString('Asserts failed: ');
	   addValue(sStatistic.u32Failed);

	7: //

	9:  addString('Ergebnis : ');
		IF sStatistic.u32Failed > 0 THEN
			addString('FAILED');
		ELSE
			addString('PASSED');
		END_IF;

	10: addString('++++++++++++++++++++++++++++++++++++++++++++++++++');
	
	99: BuildFile := ERetCode_t.eRetDone;

	END_CASE;
END_METHOD

(******************************************************************************
Baustein: FB_TestReportBase.getFileName
Spezifikation: doc/Spezifikation.pdf, Kap. x.y.z
-------------------------------------------------------------------------------
erstellt:
von:
Geändert:
von:
-------------------------------------------------------------------------------
Beschreibung
Diese Methode muss vom ableitenden Baustein überschrieben werden und
wird von der Basisklasse aus aufgerufen wenn der Report erstellt werden
soll.

-------------------------------------------------------------------------------
Input
-

Output
-
******************************************************************************)
METHOD PROTECTED getFileName : ERetCode_t
VAR_INPUT
	i_pFileName : NameHandle_t;
	i_pPath		: PathHandle_t;
END_VAR
VAR
	sTime : TIMESTRUCT;
END_VAR

	i_pFileName^ := 'Exp_';
	i_pPath^ 	 := 'C:\Users\Administrator\Desktop\TestResult\';

	sTime := getTime();

	i_pFileName^ := Concat(i_pFileName^, WORD_TO_STRING(sTime.wYear));
	i_pFileName^ := Concat(i_pFileName^, DWORD_TO_DECSTR(sTime.wMonth, 2));
	i_pFileName^ := Concat(i_pFileName^, DWORD_TO_DECSTR(sTime.wDay  , 2));
	i_pFileName^ := Concat(i_pFileName^, '_');
	i_pFileName^ := Concat(i_pFileName^, DWORD_TO_DECSTR(sTime.wHour  , 2));
	i_pFileName^ := Concat(i_pFileName^, DWORD_TO_DECSTR(sTime.wMinute, 2));
	i_pFileName^ := Concat(i_pFileName^, '.txt');
END_METHOD

END_FUNCTION_BLOCK
